INTERFACE I_EtherCATDevice

METHOD IsDeviceOK : BOOL
VAR_INPUT
END_VAR
END_METHOD

END_INTERFACE

(* stored: Version 1.1.0.1, ProductVersion 3.1.4024.12
   Itf I_EtherCATDevice: Id {f234e03e-fdb2-43fa-b3d9-a8e372931485}
   Method IsDeviceOK: Id {c799f040-fc1d-4517-bebc-2e881256725b} *)
